// TIA Portal V20 export
// export: Created 2025-12-01T14:57:11.1564012Z, ExportSetting None, DisplayName Totally Integrated Automation Portal, DisplayVersion V20 Update 3, DisplayName TIA Portal Openness, DisplayVersion V20 Update 3, DisplayName TIA Portal Version Control Interface, DisplayVersion V20 Update 3, DisplayName STEP 7 Professional, DisplayVersion V20 Update 3, DisplayName STEP 7 Safety, DisplayVersion V20 Update 2, DisplayName WinCC Basic/Comfort/Advanced, DisplayVersion V20 Update 3, DisplayName WinCC Professional, DisplayVersion V20 Update 3, DisplayName WinCC Unified, DisplayVersion V20 Update 3
FUNCTION "FC819_EventosEnv_CambiarUTDeMesa" : Void   // FC819, STL
TITLE = Emision de los Eventos del la Etiquetadora
{ S7_Optimized_Access := 'FALSE' }
AUTHOR : TRACKING
NAME : 20141014
VERSION : 4.1
// stored: AutoNumber false
   VAR_INPUT
      NumeroUT : UInt;   // Numero de Maquina
      MesaPantalla : UInt;
      MesaDestino : UInt;
   END_VAR
   VAR_TEMP
      P_EmiEventos : DWord;
      DBEventos : Word;
      NumDBEventos : UInt;
      MaxBytes : UInt;
      NumBytes : UInt;
      MesaTMP : UInt;
      DestinoDelCambio : UInt;
      NumUTsEnOrigen : UInt;
      NumUTsEnDestino : UInt;
      PosicionDeLaUT : UInt;
      SiguienteUT : UInt;
      OffsetInicial : UInt;
      OffsetFinal : UInt;
      Valor : UDInt;
   END_VAR
BEGIN

NETWORK
TITLE = Inicializaciones
///////////////////////////////////////////////////////////////////////////////
/// Mirar Si pertenece al JDT 02 (Por Defecto JDT01)

      L     "JDT1_NDB_EventosEmi";
      T     #DBEventos;
      T     #NumDBEventos;
      L     "JDT1_MaxBytes";
      T     #MaxBytes;

      SET;
      AN    "DB850_DefinicionMesas".Mesa[#MesaPantalla].ConfigMesa.MesaDeJDT02;
      JC    NoPerteneceJdT02;

      L     "JDT2_NDB_EventosEmi";
      T     #DBEventos;
      T     #NumDBEventos;
      L     "JDT2_MaxBytes";
      T     #MaxBytes;

NoPerteneceJdT02:NOP   0;

/// Final --> Pertenece al JDT 02
///////////////////////////////////////////////////////////////////////////////



NETWORK
TITLE = Mirar si se pueden generar eventos
// - Inicializo el Numero de Bytes y el puntero del DB de Eventos Generados
// - Calcula el Tamaño de bytes que hay en el DB de Eventos Genardos
// - Comprobamos si hay sitio para Eventos
///////////////////////////////////////////////////////////////////////////////
// Inicializo el Numero de Bytes y el puntero del DB Eventos Generados

      L     0;
      T     #NumBytes;  // Inicializo el numero de Bytes
      LAR2;  // Inicializo el puntero de Eventos Generados

///////////////////////////////////////////////////////////////////////////////
// Calcula el tamaño de bytes que hay en el DB Eventos Generados

      OPN   DB [#DBEventos];

Inicio_BusquedaFinalEventos:NOP   0;
      L     DBB [AR2, P#0.0];
      L     0;
      ==I;
      JC    Fin_BusquedaFinalEventos;  // Buscamos el final del DB = 0

      +AR2  P#1.0;
      JU    Inicio_BusquedaFinalEventos;

Fin_BusquedaFinalEventos:NOP   0;
      TAR2;  // Guardo el puntero
      T     #P_EmiEventos;  // Sacamos el NumBytes Escritos
      SRD   3;
      T     #NumBytes;

///////////////////////////////////////////////////////////////////////////////
// Comprobamos si hay sitio para mas Eventos

      L     #NumBytes;  // Miramos si hay sitio
      L     #MaxBytes;  // Max. que se pueden emitir, parametro
      >I;
      JC    FinalFuncion;  // No se pueden generar más eventos



NETWORK
TITLE = Recoger Datos --> Para el Formateo del Evento
///////////////////////////////////////////////////////////////////////////////
/// Calculo de Numero de Bytes en Origen y En destino

      CALL  "FC871_NumUTsEnMesa"
      ( Mesa   := #MesaPantalla,
        NumUTs := #NumUTsEnOrigen
      );

      L     #MesaDestino;
      L     "CTE_OffsetMesa";
      -I;
      T     #MesaTMP;
      CALL  "FC871_NumUTsEnMesa"
      ( Mesa   := #MesaTMP,
        NumUTs := #NumUTsEnDestino
      );


///////////////////////////////////////////////////////////////////////////////
/// Recoger Datos de la UT --> Formateo del Evento

      L     #MesaDestino;
      T     #DestinoDelCambio;


/// Calculo de la Posicion de la UT

      L     "DB810_ColasMesas".Colas[#MesaPantalla].UT_PrimeraMesa;
      T     #SiguienteUT;

      L     1;  // Siempre hay una UT en la Mesa
      T     #PosicionDeLaUT;

InicioCalculoPosicion:NOP   0;
      L     #NumeroUT;  // Es la UT que se busca
      L     #SiguienteUT;
      ==I;
      JC    FinCalculoPosicion;

      L     #PosicionDeLaUT;  // Incremento de Posicion
      L     1;
      +I;
      T     #PosicionDeLaUT;

      L     "DB812_UTs_Control".UT[#SiguienteUT].UT_SiguienteMesa;
      T     #SiguienteUT;
      JU    InicioCalculoPosicion;

FinCalculoPosicion:NOP   0;
      JU    EmitirEvento_PeticionCambiarUTDeMesa;



NETWORK
TITLE = Emision del Evento
EmitirEvento_PeticionCambiarUTDeMesa:NOP   0;

///////////////////////////////////////////////////////////////////////////////
// --- Formateo del Evento PROC - Estado del Proceso de la Maquina

      L     #P_EmiEventos;
      LAR2;  // Puntero al DB de Eventos Generados

      TAR2;  // Mirar si es el primer evento de la lista
      L     0;
      ==I;
      JC    NoEsInicio_ListaDeEventos;  // Es el primero

      OPN   DB [#DBEventos];
      L     ',';  // Separador entre eventos ','
      T     DBB [AR2, P#0.0];
      +AR2  P#1.0;

NoEsInicio_ListaDeEventos:NOP   0;

///////////////////////////////////////////////////////////////////////////////
// --- Cuerpo del Evento

      OPN   DB [#DBEventos];  // DB de Eventos Generados (A Emitir)
      L     '{';  // Inicio de Evento '{'
      T     DBB [AR2, P#0.0];
      +AR2  P#1.0;

      L     'MOV?';  // Evento 'DATO'
      T     DBD [AR2, P#0.0];
      +AR2  P#4.0;


///////////////////////////////////////////////////////////////////////////////
      L     '[';  // Evento - Atributo MCKY '[MCKY]'
      T     DBB [AR2, P#0.0];
      L     'MCKY';
      T     DBD [AR2, P#1.0];
      L     ']';
      T     DBB [AR2, P#5.0];
      +AR2  P#6.0;

// --- Convertir Valor a ASCII - Mckey
      TAR2;
      SRD   3;
      T     #OffsetInicial;  // Miro que offset tiene la String

      L     "DB812_UTs_Control".UT[#NumeroUT].Mckey;
      T     #Valor;

      CALL  "FC893_Obtener_StringDelAtributo"
      ( DB_String := #NumDBEventos,
        OffsetIni := #OffsetInicial,
        Valor     := #Valor,
        OffsetFin := #OffsetFinal
      );  // Llamo a ObtenerStrinAtributo

      L     #OffsetFinal;
      SLD   3;
      LAR2;  // Recupero que offset tiene la String

// --- Ya esta convertido el Valor a ASCI - Fin Mckey


///////////////////////////////////////////////////////////////////////////////
      OPN   DB [#DBEventos];  // DB de Eventos Generados (A Emitir)
      L     '[';  // Evento - Atributo MESA '[MESA]'
      T     DBB [AR2, P#0.0];
      L     'MESA';
      T     DBD [AR2, P#1.0];
      L     ']';
      T     DBB [AR2, P#5.0];
      +AR2  P#6.0;

// --- Convertir Valor a ASCII - Numero de Mesa
      TAR2;
      SRD   3;
      T     #OffsetInicial;  // Miro que offset tiene la String

      L     "DB812_UTs_Control".UT[#NumeroUT].MesaActual;
      T     #Valor;

      CALL  "FC893_Obtener_StringDelAtributo"
      ( DB_String := #NumDBEventos,
        OffsetIni := #OffsetInicial,
        Valor     := #Valor,
        OffsetFin := #OffsetFinal
      );  // Llamo a ObtenerStrinAtributo

      L     #OffsetFinal;
      SLD   3;
      LAR2;  // Recupero que offset tiene la String

// --- Ya esta convertido el Valor a ASCI - Numero de Mesa


///////////////////////////////////////////////////////////////////////////////
      OPN   DB [#DBEventos];  // DB de Eventos Generados (A Emitir)
      L     '[';  // Evento - Atributo POSICION '[POSI]'
      T     DBB [AR2, P#0.0];
      L     'POSI';
      T     DBD [AR2, P#1.0];
      L     ']';
      T     DBB [AR2, P#5.0];
      +AR2  P#6.0;

// --- Convertir Valor a ASCII - Numero de Posicion
      TAR2;
      SRD   3;
      T     #OffsetInicial;  // Miro que offset tiene la String

      L     #PosicionDeLaUT;
      T     #Valor;

      CALL  "FC893_Obtener_StringDelAtributo"
      ( DB_String := #NumDBEventos,
        OffsetIni := #OffsetInicial,
        Valor     := #Valor,
        OffsetFin := #OffsetFinal
      );  // Llamo a ObtenerStrinAtributo

      L     #OffsetFinal;
      SLD   3;
      LAR2;  // Recupero que offset tiene la String

// --- Ya esta convertido el Valor a ASCI - Numero de Posicion


///////////////////////////////////////////////////////////////////////////////
      OPN   DB [#DBEventos];  // DB de Eventos Generados (A Emitir)
      L     '[';  // Evento - Atributo DESTINO '[DEST]'
      T     DBB [AR2, P#0.0];
      L     'DEST';
      T     DBD [AR2, P#1.0];
      L     ']';
      T     DBB [AR2, P#5.0];
      +AR2  P#6.0;

// --- Convertir Valor a ASCII - Numero de Destino
      TAR2;
      SRD   3;
      T     #OffsetInicial;  // Miro que offset tiene la String

      L     #DestinoDelCambio;
      T     #Valor;

      CALL  "FC893_Obtener_StringDelAtributo"
      ( DB_String := #NumDBEventos,
        OffsetIni := #OffsetInicial,
        Valor     := #Valor,
        OffsetFin := #OffsetFinal
      );  // Llamo a ObtenerStrinAtributo

      L     #OffsetFinal;
      SLD   3;
      LAR2;  // Recupero que offset tiene la String

// --- Ya esta convertido el Valor a ASCI - Numero de Destino


///////////////////////////////////////////////////////////////////////////////
      OPN   DB [#DBEventos];  // DB de Eventos Generados (A Emitir)
      L     '[';  // Evento - Atributo NUMERO DE UTS EN ORIGEN '[CORG]'
      T     DBB [AR2, P#0.0];
      L     'CORG';
      T     DBD [AR2, P#1.0];
      L     ']';
      T     DBB [AR2, P#5.0];
      +AR2  P#6.0;

// --- Convertir Valor a ASCII - Numero de UTs en Origen
      TAR2;
      SRD   3;
      T     #OffsetInicial;  // Miro que offset tiene la String

      L     #NumUTsEnOrigen;
      T     #Valor;

      CALL  "FC893_Obtener_StringDelAtributo"
      ( DB_String := #NumDBEventos,
        OffsetIni := #OffsetInicial,
        Valor     := #Valor,
        OffsetFin := #OffsetFinal
      );  // Llamo a ObtenerStrinAtributo

      L     #OffsetFinal;
      SLD   3;
      LAR2;  // Recupero que offset tiene la String

// --- Ya esta convertido el Valor a ASCI - Numero de UTs en Origen


///////////////////////////////////////////////////////////////////////////////
      OPN   DB [#DBEventos];  // DB de Eventos Generados (A Emitir)
      L     '[';  // Evento - Atributo NUMERO DE UTS EN DESTINO '[CDST]'
      T     DBB [AR2, P#0.0];
      L     'CDST';
      T     DBD [AR2, P#1.0];
      L     ']';
      T     DBB [AR2, P#5.0];
      +AR2  P#6.0;

// --- Convertir Valor a ASCII - Numero de UTs en Destino
      TAR2;
      SRD   3;
      T     #OffsetInicial;  // Miro que offset tiene la String

      L     #NumUTsEnDestino;
      T     #Valor;

      CALL  "FC893_Obtener_StringDelAtributo"
      ( DB_String := #NumDBEventos,
        OffsetIni := #OffsetInicial,
        Valor     := #Valor,
        OffsetFin := #OffsetFinal
      );  // Llamo a ObtenerStrinAtributo

      L     #OffsetFinal;
      SLD   3;
      LAR2;  // Recupero que offset tiene la String

// --- Ya esta convertido el Valor a ASCI - Numero de UTs en Destino





///////////////////////////////////////////////////////////////////////////////
// --- Final del formateo del Evento

      OPN   DB [#DBEventos];  // DB de Eventos Generados (A Emitir)
      L     '}';  // Fin de Evento '}'
      T     DBB [AR2, P#0.0];
      +AR2  P#1.0;

///////////////////////////////////////////////////////////////////////////////
// --- Dar por formateado el Evento

      SET;
      S     "DB812_UTs_Control".UT[#NumeroUT].EventosDeCambioDeMesa.PeticionCambiarUTDeMesa;

      JU    FinalFuncion;  // Ya se ha generado el evento de la Maquina

// --- Fin del Formateo del Evento de Estado del Proceso
///////////////////////////////////////////////////////////////////////////////



NETWORK
TITLE = Fin de la Funcion
///////////////////////////////////////////////////////////////////////////////
// --- Final de la función
FinalFuncion:NOP   0;


END_FUNCTION
